PROGRAM prgHouse
VAR
	fbKBusState					: FB_K_Bus_State;
	uint_KBusState				: UINT;							
	lrHousePower				: LREAL;								
	lrNetzEinspeisung			: LREAL;								
	lrBetriebMuellerBau			: LREAL;								
	fbGrid1						: FB_EM_Beckhoff_KL3403;  	//UV Müller Holzbau
	fbGrid2						: FB_EM_Beckhoff_KL3403;	//Abgang Direktmessung
	fbGrid3						: FB_EM_Beckhoff_KL3403;	//Produktion PV
	(*
	lrGrid_Voltage_L1  	AT %I* : LREAL;										
    lrGrid_Current_L1 	AT %I* : LREAL;	
	lrGrid_Power_L1		AT %I* : LREAL;		
	lrGrid_Voltage_L2  	AT %I* : LREAL;										
    lrGrid_Current_L2 	AT %I* : LREAL;	
	lrGrid_Power_L2		AT %I* : LREAL;
	lrGrid_Voltage_L3  	AT %I* : LREAL;										
    lrGrid_Current_L3 	AT %I* : LREAL;	
	lrGrid_Power_L3		AT %I* : LREAL;									
	ActivePowerTotal	AT %I* : LREAL;		
	Test					   : REAL;	
*)
	lrGrid_Voltage_L1  	AT %I* 	: REAL;										
    lrGrid_Current_L1 	AT %I* 	: REAL;	
	lrGrid_Power_L1		AT %I* 	: REAL;		
	lrGrid_Voltage_L2  	AT %I* 	: REAL;										
    lrGrid_Current_L2 	AT %I* 	: REAL;	
	lrGrid_Power_L2		AT %I* 	: REAL;
	lrGrid_Voltage_L3  	AT %I* 	: REAL;										
    lrGrid_Current_L3 	AT %I* 	: REAL;	
	lrGrid_Power_L3		AT %I* 	: REAL;									
	ActivePowerTotal	AT %I*	: REAL;							
								
END_VAR

//lrNetzEinspeisung := fbGrid1.stDataEMPower.lrPowerTotal + fbGrid2.stDataEMPower.lrPowerTotal - fbGrid3.stDataEMPower.lrPowerTotal;	

//lrBetriebMuellerBau := (ActivePowerTotal_1 + ActivePowerTotal_2 + ActivePowerTotal_3) - fbGrid1.stDataEMPower.lrPowerTotal;

//The mapping of this function must be linked with the K-Bus State in the E/A Part
fbKBusState(	uiKBusState_OUT=> , 
				b_Kbus_notOk=> , 
				word_ErrorCount=> );
				
				


(*
fbGrid1(
	bEnable:= FALSE, 
	bChannel1Invers:= FALSE, 
	bChannel2Invers:= FALSE, 
	bChannel3Invers:= FALSE, 
	uiCurrentTransformerRatioL1:= 400, 
	uiCurrentTransformerRatioL2:= 400, 
	uiCurrentTransformerRatioL3:= 400, 
	uiKBusState_IN:= fbKBusState.uiKBusState_OUT, 
	stDataEMPower=> , 
	stDataEMCounter=> , 
	stDataEMPowerRealTime=> , 
	stDataEMCounterRealTime=> , 
	diNrOfEM_OUT=> );
	
	
fbGrid2(
	bEnable:= FALSE, 
	bChannel1Invers:= FALSE, 
	bChannel2Invers:= FALSE, 
	bChannel3Invers:= FALSE, 
	uiCurrentTransformerRatioL1:= 400, 
	uiCurrentTransformerRatioL2:= 400, 
	uiCurrentTransformerRatioL3:= 400, 
	uiKBusState_IN:= , 
	stDataEMPower=> , 
	stDataEMCounter=> , 
	stDataEMPowerRealTime=> , 
	stDataEMCounterRealTime=> , 
	diNrOfEM_OUT=> );
	
fbGrid3(
	bEnable:= FALSE, 
	bChannel1Invers:= FALSE, 
	bChannel2Invers:= FALSE, 
	bChannel3Invers:= FALSE, 
	uiCurrentTransformerRatioL1:= 400, 
	uiCurrentTransformerRatioL2:= 400, 
	uiCurrentTransformerRatioL3:= 400, 
	uiKBusState_IN:= , 
	stDataEMPower=> , 
	stDataEMCounter=> , 
	stDataEMPowerRealTime=> , 
	stDataEMCounterRealTime=> , 
	diNrOfEM_OUT=> );
*)

END_PROGRAM

(* stored: Version 1.1.0.1, ProductVersion 3.1.4024.13
   POU prgHouse: Id {2627c3a1-fabe-46fd-8396-cc823b8dfb91}, SpecialFunc None *)
